// Mitsubishi GX Works2 project: gg   PLC: FX3G

// global labels: Global1
VAR_GLOBAL
  startMach AT X007 : BOOL;
  machOn AT M0 : BOOL;
  senWeight AT X000 : BOOL;
  GG_placed AT M1 : BOOL;
  dropGummyBear AT X001 : BOOL;
  countGummys AT CC1 : BOOL;
END_VAR
VAR_GLOBAL CONSTANT
  counter6 : INT := 6;
END_VAR
VAR_GLOBAL
  reached6 AT CS1 : BOOL;
  finishFilling AT M2 : BOOL;
  enoughGummys AT X002 : BOOL;
  fillingOn AT Y004 : BOOL;
  senWeight2 AT X003 : BOOL;
  senWeight1 AT X004 : BOOL;
  moreGGToFill AT M3 : BOOL;
  error AT X005 : BOOL;
  runnerOn AT Y002 : BOOL;
END_VAR

// task Task_01 (event TRUE, interval 0, priority 31): POU_01

PROGRAM POU_01
(* structured ladder/FBD written out as ST: instructions are called as NAME(EN, inputs, outputs); _pN, _eN, _tN stand for wires *)
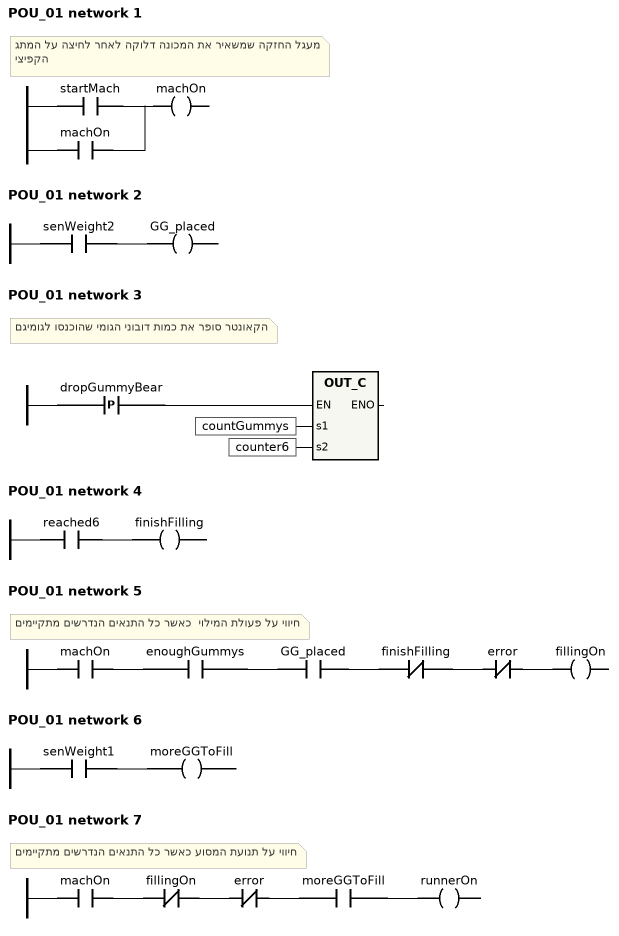
(* network 1 *)
(* מעגל החזקה שמשאיר את המכונה דלוקה לאחר לחיצה על המתג הקפיצי *)
machOn := startMach OR machOn;
(* network 2 *)
GG_placed := senWeight2;
(* network 3 *)
(* הקאונטר סופר את כמות דובוני הגומי שהוכנסו לגומיגם *)
OUT_C(LDP(TRUE, dropGummyBear), countGummys, counter6);
(* network 4 *)
finishFilling := reached6;
(* network 5 *)
(* חיווי על פעולת המילוי  כאשר כל התנאים הנדרשים מתקיימים *)
fillingOn := machOn AND enoughGummys AND GG_placed AND NOT finishFilling AND NOT error;
(* network 6 *)
moreGGToFill := senWeight1;
(* network 7 *)
(* חיווי על תנועת המסוע כאשר כל התנאים הנדרשים מתקיימים *)
runnerOn := machOn AND NOT fillingOn AND NOT error AND moreGGToFill;
END_PROGRAM
